FUNCTION_BLOCK GenericCylinderModelType2 (* Composite Function Block Type *)
  (* Standard: 61499-2 *)
  (* Version 0.0, 2/3/2012, XPMUser, nxtControl GmbH, template *)
  PACKAGE Main;
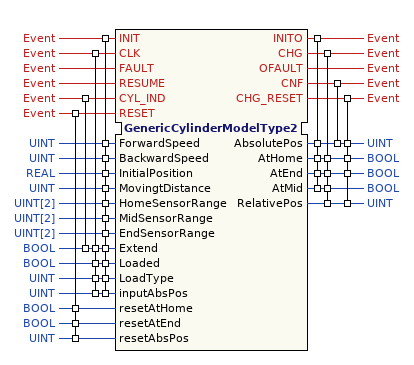
  EVENT_INPUT
    INIT WITH ForwardSpeed, BackwardSpeed, Extend, HomeSensorRange, EndSensorRange, InitialPosition, LoadType, MovingtDistance, Loaded, MidSensorRange, inputAbsPos; (* Initialization Request *)
    CLK WITH Extend, Loaded, LoadType, inputAbsPos; (* Clock signal *)
    FAULT;
    RESUME;
    CYL_IND WITH Extend;
    RESET WITH resetAtHome, resetAtEnd, resetAbsPos;
  END_EVENT
  EVENT_OUTPUT
    INITO WITH AbsolutePos, AtHome, AtEnd, AtMid; (* Initialization Confirm *)
    CHG WITH AtHome, AtEnd, AtMid, RelativePos; (* Indicate data outputs changed *)
    OFAULT;
    CNF WITH AbsolutePos;
    CHG_RESET WITH AbsolutePos, AtHome, AtEnd, RelativePos;
  END_EVENT
  VAR_INPUT
    ForwardSpeed : UINT; (* Forward speed *)
    BackwardSpeed : UINT; (* Backward speed *)
    InitialPosition : REAL; (* Initial position *)
    MovingtDistance : UINT; (* Moving distance *)
    HomeSensorRange : ARRAY [0..1] OF UINT; (* Detection range of home sensor *)
    MidSensorRange : ARRAY [0..1] OF UINT; (* Detection range of home sensor *)
    EndSensorRange : ARRAY [0..1] OF UINT; (* Detection range of end sensor *)
    Extend : BOOL;
    Loaded : BOOL;
    LoadType : UINT;
    inputAbsPos : UINT;
    resetAtHome : BOOL;
    resetAtEnd : BOOL;
    resetAbsPos : UINT;
  END_VAR
  VAR_OUTPUT
    AbsolutePos : UINT; (* Current position *)
    AtHome : BOOL; (* Detected at home position *)
    AtEnd : BOOL; (* Detected at end position *)
    AtMid : BOOL;
    RelativePos : UINT;
  END_VAR
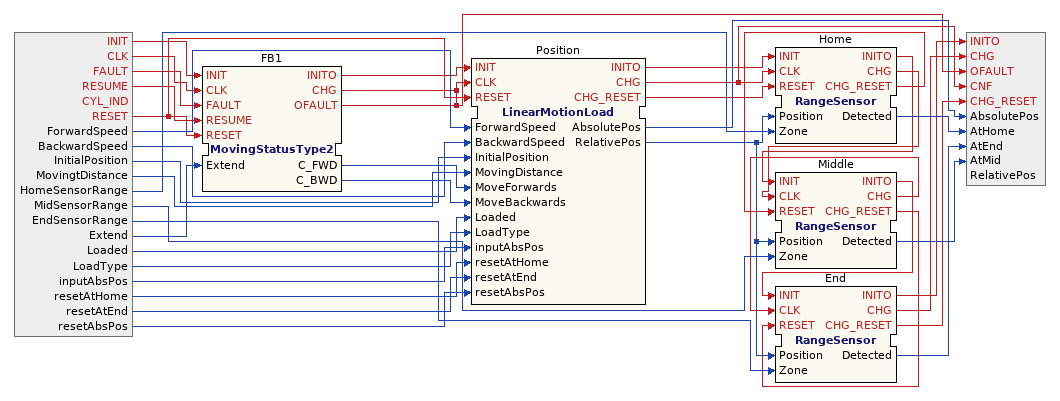
  FBS
    Home : RangeSensor;
    Middle : RangeSensor;
    End : RangeSensor;
    Position : LinearMotionLoad;
    FB1 : MovingStatusType2;
  END_FBS
  EVENT_CONNECTIONS
    Position.INITO TO Home.INIT;
    Home.INITO TO Middle.INIT;
    Middle.INITO TO End.INIT;
    End.INITO TO INITO;
    Position.CHG TO CNF;
    Position.CHG TO Home.CLK;
    INIT TO FB1.INIT;
    FAULT TO FB1.FAULT;
    RESUME TO FB1.RESUME;
    FB1.INITO TO Position.INIT;
    FB1.OFAULT TO OFAULT;
    RESET TO Position.RESET;
    Home.CHG TO Middle.CLK;
    Middle.CHG TO End.CLK;
    Home.CHG_RESET TO Middle.RESET;
    Middle.CHG_RESET TO End.RESET;
    End.CHG TO CHG;
    End.CHG_RESET TO CHG_RESET;
    Position.CHG_RESET TO Home.RESET;
    CLK TO FB1.CLK;
    FB1.CHG TO Position.CLK;
    FB1.OFAULT TO Position.CLK;
    RESET TO FB1.RESET;
  END_CONNECTIONS
  DATA_CONNECTIONS
    Loaded TO Position.Loaded;
    LoadType TO Position.LoadType;
    EndSensorRange TO End.Zone;
    HomeSensorRange TO Home.Zone;
    Position.RelativePos TO Middle.Position;
    Position.RelativePos TO End.Position;
    Home.Detected TO AtHome;
    Middle.Detected TO AtMid;
    End.Detected TO AtEnd;
    ForwardSpeed TO Position.ForwardSpeed;
    BackwardSpeed TO Position.BackwardSpeed;
    InitialPosition TO Position.InitialPosition;
    MovingtDistance TO Position.MovingDistance;
    Position.AbsolutePos TO AbsolutePos;
    Position.RelativePos TO Home.Position;
    MidSensorRange TO Middle.Zone;
    Extend TO FB1.Extend;
    inputAbsPos TO Position.inputAbsPos;
    FB1.C_FWD TO Position.MoveForwards;
    FB1.C_BWD TO Position.MoveBackwards;
    resetAtHome TO Position.resetAtHome;
    resetAtEnd TO Position.resetAtEnd;
    resetAbsPos TO Position.resetAbsPos;
  END_CONNECTIONS
END_FUNCTION_BLOCK
